INTERFACE iCalculationTask EXTENDS TcoCore.ITcoTask

PROPERTY CoordinatesInMillimeter : REFERENCE TO Coordinates
GET
END_GET
END_PROPERTY

PROPERTY DistanceFromObject : LREAL
GET
END_GET
END_PROPERTY

PROPERTY FieldOfView : REFERENCE TO FieldOfView
GET
END_GET
END_PROPERTY

END_INTERFACE

(* stored: Version 1.1.0.1, ProductVersion 3.1.4024.12
   Itf iCalculationTask: Id {8b6b9015-5792-0ecb-107e-395b86bf073d}
   Folder Data: Id {8228426c-ab5b-0602-2da6-6b33d8775a71}
   Property CoordinatesInMillimeter: Id {04b3ef71-22c7-0d43-37ae-9edd28b36a9f}
   Get Get: Id {48266f35-de7f-0b7d-02d7-3afdded76614}
   Property DistanceFromObject: Id {cfbed818-91b8-094a-1fca-feb1779430ec}
   Get Get: Id {6193bb55-0e72-0afb-16cc-5511227aeb88}
   Property FieldOfView: Id {c468fd7f-5bc5-0760-0090-ce1e45411134}
   Get Get: Id {1eda54fb-ecb2-0b7f-280f-019eee84e5a3} *)
